FUNCTION_BLOCK REGRESS (* Single-Variable Linear Time Series Regression *)
  (* Standard: IEC 61499-1; Classification: Math; ApplicationDomain: General; Function: Linear Regression; Type: Single Time Series; Description: Single-variable linear time series regression *)
  (* Version 0.0, 2006-04-28, JHC, Holobloc Inc *)
  (* Compiler header: package fb.rt.math; *)
  (* Compiler Java Sun JDK 1.5.0 *)
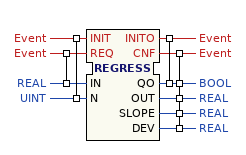
  EVENT_INPUT
    INIT WITH N; (* Set N, reset outputs and sample buffer *)
    REQ WITH IN; (* Sample Clock, Uniform Interval *)
  END_EVENT
  EVENT_OUTPUT
    INITO WITH QO; (* Initialization Confirm *)
    CNF WITH QO, OUT, SLOPE, DEV; (* Execution Confirmation *)
  END_EVENT
  VAR_INPUT
    IN : REAL; (* Sampled Variable *)
    N : UINT := 16; (* Number of samples in series *)
  END_VAR
  VAR_OUTPUT
    QO : BOOL; (* Sample buffer full, outputs valid *)
    OUT : REAL; (* Projected next value of IN *)
    SLOPE : REAL; (* Slope of regressed data, IN units per clock period. *)
    DEV : REAL; (* Estimated standard deviation from regression line *)
  END_VAR
END_FUNCTION_BLOCK
